Staubli VAL3: MainKey.pgx

program MainKey(num x_nKey)
  local num l_nKey
begin

  switch x_nKey
    //砂带初始化
    case 271
      call OnF1()
    break
    //坐标整体偏移
    case 272
      call OnF2()
    break
    //记录
    case 273
      call OnF3()
    break
    //运行
    case 274
      taskSuspend("Move2P")
      call OnF4()
      taskResume("Move2P",0)
    break
    //
    case 275
    break
    //重载数据
    case 276
      call OnF6()
    break
    //保存
    case 277
      call OnF7()
    break
  endSwitch
end
